// TIA Portal V16 export
// export: Created 2022-11-17T15:49:26.75894Z, ExportSetting WithDefaults, DisplayName Totally Integrated Automation Portal, DisplayVersion V16 Update 6, DisplayName TIA Portal Version Control Interface, DisplayVersion V16 Update 2, DisplayName TIA Portal Openness, DisplayVersion V16 Update 6, DisplayName SINAMICS Startdrive Advanced, DisplayVersion V16 Update 5, DisplayName SINAMICS Startdrive G130, G150, S120, S150, SINAMICS MV, S210, DisplayVersion V16 Update 5, DisplayName SINAMICS Startdrive G110M, G120, G120C, G120D, G120P, G115D, DisplayVersion V16 Update 5, DisplayName STEP 7 Professional, DisplayVersion V16 Update 6, DisplayName STEP 7 Safety, DisplayVersion V16, DisplayName WinCC Advanced, DisplayVersion V16 Update 6
FUNCTION "FC58_TableRotationPos" : Void   // FC58, LAD
{ S7_Optimized_Access := 'FALSE' }
VERSION : 0.1
// stored: AutoNumber false, IsIECCheckEnabled false, SetENOAutomatically false, UDAEnableTagReadback false
   VAR_INPUT
      PHASE : Bool;
   END_VAR
   VAR_TEMP
      TempDInt3 : DInt;
      PulseOffset : DInt;
      AC1 : Real;
      AC2 : Real;
      AC3 : Real;
      DeltaV : Real;
      DeltaVMax : Real;
      VattpiuVmin : Real;
      VmaxpiuVmin : Real;
      AC1_INT : Int;
      PulseReset : Bool;
      TEMPOMAX : Real;
      TEMPO : Real;
      Encoder : Int;
      TempDint : DInt;
      TempInt : Int;
      TempDint2 : DInt;
      TempDInt4 : DInt;
      TempWord : Word;
   END_VAR
   VAR_TEMP   // added for the SCL form of the ladder/FBD networks
      _w1 : Bool;
   END_VAR
BEGIN

REGION Network 1
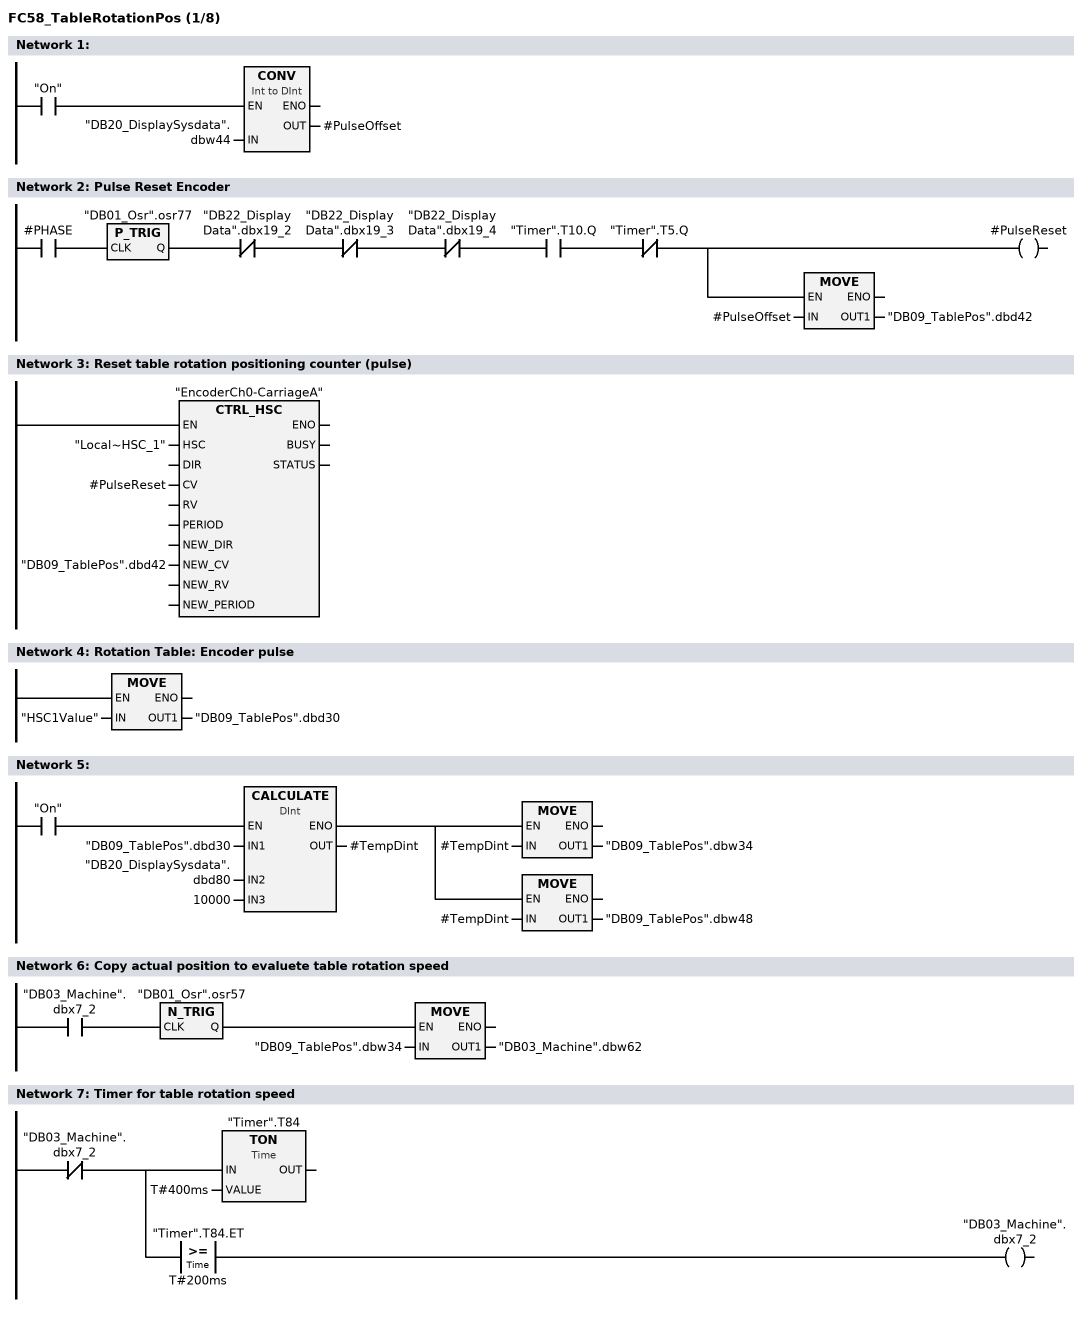
   RUNG wire#powerrail
      Contact( "On" )
      { S7_Templates := "[SrcType := Int, DestType := DInt]"; S7_GenerateENO := "TRUE" } Convert(in := "DB20_DisplaySysdata".dbw44, out => #PulseOffset)
   END_RUNG
   // the same network as SCL:
   IF "On" THEN #PulseOffset := INT_TO_DINT("DB20_DisplaySysdata".dbw44); END_IF;
END_REGION

REGION Network 2: Pulse Reset Encoder
   RUNG wire#powerrail
      Contact( #PHASE )
      P_Trig( "DB01_Osr".osr77 )
      I_Contact( "DB22_DisplayData".dbx19_2 )
      I_Contact( "DB22_DisplayData".dbx19_3 )
      I_Contact( "DB22_DisplayData".dbx19_4 )
      Contact( "Timer".T10.Q )
      I_Contact( "Timer".T5.Q )
      wire#w1
      Coil( #PulseReset )
   END_RUNG
   RUNG wire#w1
      { S7_GenerateENO := "TRUE" } Move(in := #PulseOffset, out1 => "DB09_TablePos".dbd42)
   END_RUNG
   // the same network as SCL:
   #_w1 := #PHASE AND NOT "DB01_Osr".osr77;   // rising edge
   "DB01_Osr".osr77 := #PHASE;
   #PulseReset := #_w1 AND NOT "DB22_DisplayData".dbx19_2 AND NOT "DB22_DisplayData".dbx19_3 AND NOT "DB22_DisplayData".dbx19_4 AND "Timer".T10.Q AND NOT "Timer".T5.Q;
   IF #PulseReset THEN "DB09_TablePos".dbd42 := #PulseOffset; END_IF;
END_REGION

REGION Network 3: Reset table rotation positioning counter (pulse)
   RUNG wire#powerrail
      "EncoderCh0-CarriageA".CTRL_HSC(HSC := "Local~HSC_1", DIR :=, CV := #PulseReset, RV :=, PERIOD :=, NEW_DIR :=, NEW_CV := "DB09_TablePos".dbd42, NEW_RV :=, NEW_PERIOD :=, BUSY =>, STATUS =>)
   END_RUNG
   // the same network as SCL:
   "EncoderCh0-CarriageA"(HSC := "Local~HSC_1", CV := #PulseReset, NEW_CV := "DB09_TablePos".dbd42);   // CTRL_HSC
END_REGION

REGION Network 4: Rotation Table: Encoder pulse
   RUNG wire#powerrail
      { S7_GenerateENO := "TRUE" } Move(in := "HSC1Value", out1 => "DB09_TablePos".dbd30)
   END_RUNG
   // the same network as SCL:
   "DB09_TablePos".dbd30 := "HSC1Value";
END_REGION

REGION Network 5
   RUNG wire#powerrail
      Contact( "On" )
      { S7_Templates := "SrcType := DInt"; S7_GenerateENO := "TRUE"; S7_Expression := "((In1*In2)/In3)" } Calculate(in1 := "DB09_TablePos".dbd30, in2 := "DB20_DisplaySysdata".dbd80, in3 := 10000, out => #TempDint)
      wire#w1
      { S7_GenerateENO := "TRUE" } Move(in := #TempDint, out1 => "DB09_TablePos".dbw34)
   END_RUNG
   RUNG wire#w1
      { S7_GenerateENO := "TRUE" } Move(in := #TempDint, out1 => "DB09_TablePos".dbw48)
   END_RUNG
   // the same network as SCL:
   // ENO of a box is taken as its EN; it also drops when the box reports an error
   IF "On" THEN
       #TempDint := (("DB09_TablePos".dbd30*"DB20_DisplaySysdata".dbd80)/10000);
       "DB09_TablePos".dbw34 := #TempDint;
       "DB09_TablePos".dbw48 := #TempDint;
   END_IF;
END_REGION

REGION Network 6: Copy actual position to evaluete table rotation speed
   RUNG wire#powerrail
      Contact( "DB03_Machine".dbx7_2 )
      N_Trig( "DB01_Osr".osr57 )
      { S7_GenerateENO := "TRUE" } Move(in := "DB09_TablePos".dbw34, out1 => "DB03_Machine".dbw62)
   END_RUNG
   // the same network as SCL:
   #_w1 := NOT "DB03_Machine".dbx7_2 AND "DB01_Osr".osr57;   // falling edge
   "DB01_Osr".osr57 := "DB03_Machine".dbx7_2;
   IF #_w1 THEN "DB03_Machine".dbw62 := "DB09_TablePos".dbw34; END_IF;
END_REGION

REGION Network 7: Timer for table rotation speed
   #_w1 := NOT "DB03_Machine".dbx7_2;
   "Timer".T84.TON(IN := #_w1, PT := T#400ms);   // TON coil
   "DB03_Machine".dbx7_2 := #_w1 AND ("Timer".T84.ET >= T#200ms);
END_REGION

REGION Network 8: Speed calculation (1)
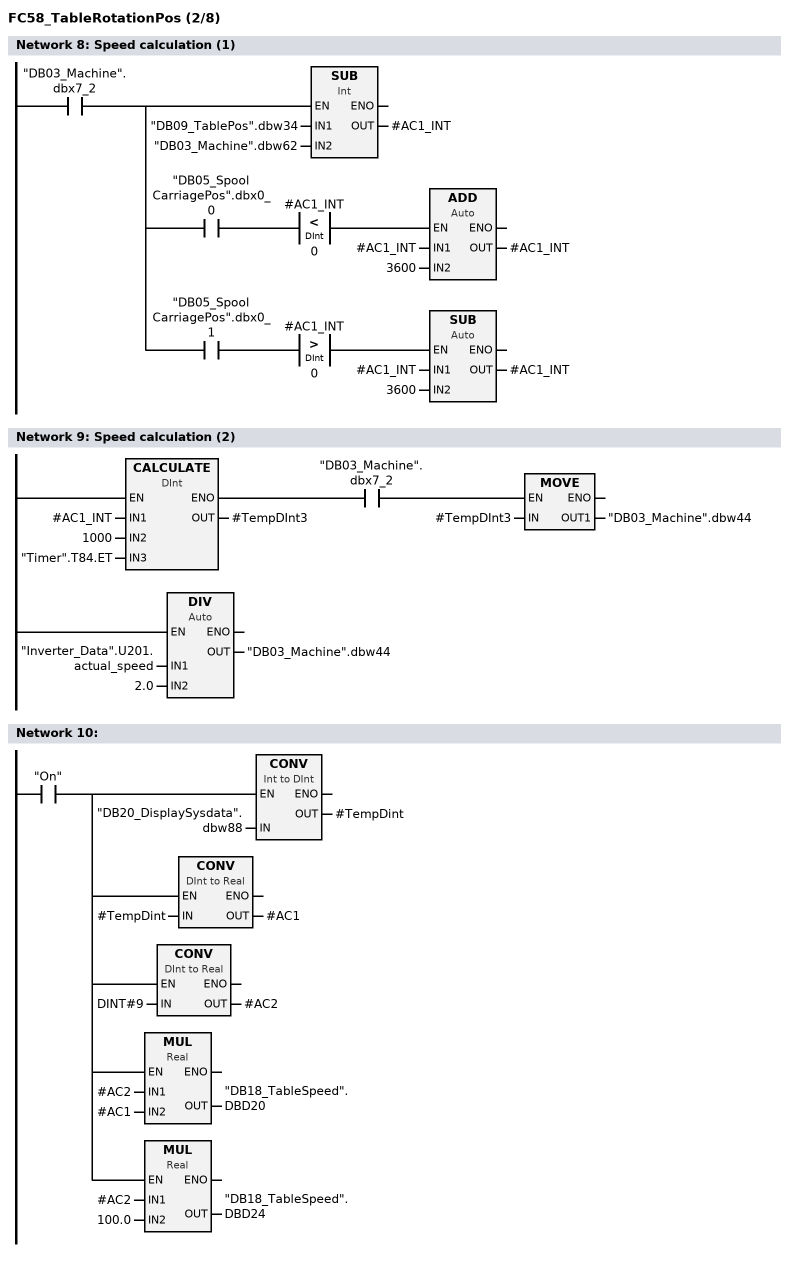
   RUNG wire#powerrail
      Contact( "DB03_Machine".dbx7_2 )
      wire#w1
      { S7_Templates := "SrcType := Int"; S7_GenerateENO := "TRUE" } Sub(in1 := "DB09_TablePos".dbw34, in2 := "DB03_Machine".dbw62, out => #AC1_INT)
   END_RUNG
   RUNG wire#w1
      Contact( "DB05_SpoolCarriagePos".dbx0_0 )
      { S7_Templates := "SrcType := DInt" } LT_Contact(in1 := #AC1_INT, in2 := 0)
      { S7_GenerateENO := "TRUE" } Add(in1 := #AC1_INT, in2 := 3600, out => #AC1_INT)
   END_RUNG
   RUNG wire#w1
      Contact( "DB05_SpoolCarriagePos".dbx0_1 )
      { S7_Templates := "SrcType := DInt" } GT_Contact(in1 := #AC1_INT, in2 := 0)
      { S7_GenerateENO := "TRUE" } Sub(in1 := #AC1_INT, in2 := 3600, out => #AC1_INT)
   END_RUNG
   // the same network as SCL:
   IF "DB03_Machine".dbx7_2 THEN #AC1_INT := "DB09_TablePos".dbw34 - "DB03_Machine".dbw62; END_IF;
   IF "DB03_Machine".dbx7_2 AND "DB05_SpoolCarriagePos".dbx0_0 AND (#AC1_INT < 0) THEN
       #AC1_INT := #AC1_INT + 3600;
   END_IF;
   IF "DB03_Machine".dbx7_2 AND "DB05_SpoolCarriagePos".dbx0_1 AND (#AC1_INT > 0) THEN
       #AC1_INT := #AC1_INT - 3600;
   END_IF;
END_REGION

REGION Network 9: Speed calculation (2)
   RUNG wire#powerrail
      { S7_Templates := "SrcType := DInt"; S7_GenerateENO := "TRUE"; S7_Expression := "((In1*In2)/In3)" } Calculate(in1 := #AC1_INT, in2 := 1000, in3 := "Timer".T84.ET, out => #TempDInt3)
      Contact( "DB03_Machine".dbx7_2 )
      { S7_GenerateENO := "TRUE" } Move(in := #TempDInt3, out1 => "DB03_Machine".dbw44)
   END_RUNG
   RUNG wire#powerrail
      Div(in1 := "Inverter_Data".U201.actual_speed, in2 := 2.0, out => "DB03_Machine".dbw44)
   END_RUNG
   // the same network as SCL:
   // ENO of a box is taken as its EN; it also drops when the box reports an error
   #TempDInt3 := ((#AC1_INT*1000)/"Timer".T84.ET);
   IF "DB03_Machine".dbx7_2 THEN "DB03_Machine".dbw44 := #TempDInt3; END_IF;
   "DB03_Machine".dbw44 := "Inverter_Data".U201.actual_speed / 2.0;
END_REGION

REGION Network 10
   RUNG wire#powerrail
      Contact( "On" )
      wire#w1
      { S7_Templates := "[SrcType := Int, DestType := DInt]"; S7_GenerateENO := "TRUE" } Convert(in := "DB20_DisplaySysdata".dbw88, out => #TempDint)
   END_RUNG
   RUNG wire#w1
      { S7_Templates := "[SrcType := DInt, DestType := Real]"; S7_GenerateENO := "TRUE" } Convert(in := #TempDint, out => #AC1)
   END_RUNG
   RUNG wire#w1
      { S7_Templates := "[SrcType := DInt, DestType := Real]"; S7_GenerateENO := "TRUE" } Convert(in := DINT#9, out => #AC2)
   END_RUNG
   RUNG wire#w1
      { S7_Templates := "SrcType := Real"; S7_GenerateENO := "TRUE" } Mul(in1 := #AC2, in2 := #AC1, out => "DB18_TableSpeed".DBD20)
   END_RUNG
   RUNG wire#w1
      { S7_Templates := "SrcType := Real"; S7_GenerateENO := "TRUE" } Mul(in1 := #AC2, in2 := 100.0, out => "DB18_TableSpeed".DBD24)
   END_RUNG
   // the same network as SCL:
   IF "On" THEN
       #TempDint := INT_TO_DINT("DB20_DisplaySysdata".dbw88);
       #AC1 := DINT_TO_REAL(#TempDint);
       #AC2 := DINT_TO_REAL(DINT#9);
       "DB18_TableSpeed".DBD20 := #AC2 * #AC1;
       "DB18_TableSpeed".DBD24 := #AC2 * 100.0;
   END_IF;
END_REGION

REGION Network 11
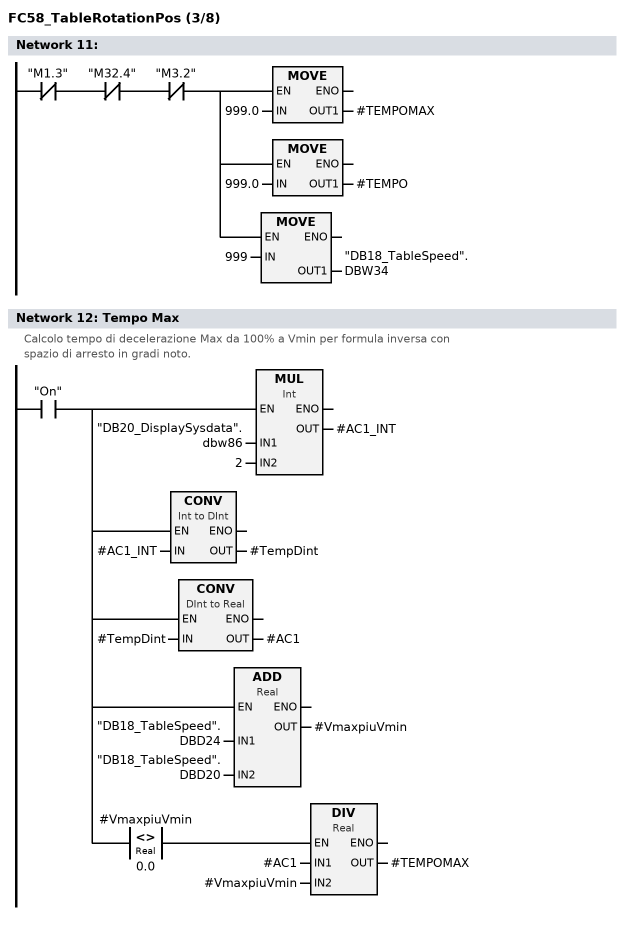
   RUNG wire#powerrail
      I_Contact( "M1.3" )
      I_Contact( "M32.4" )
      I_Contact( "M3.2" )
      wire#w1
      { S7_GenerateENO := "TRUE" } Move(in := 999.0, out1 => #TEMPOMAX)
   END_RUNG
   RUNG wire#w1
      { S7_GenerateENO := "TRUE" } Move(in := 999.0, out1 => #TEMPO)
   END_RUNG
   RUNG wire#w1
      { S7_GenerateENO := "TRUE" } Move(in := 999, out1 => "DB18_TableSpeed".DBW34)
   END_RUNG
   // the same network as SCL:
   IF NOT "M1.3" AND NOT "M32.4" AND NOT "M3.2" THEN
       #TEMPOMAX := 999.0;
       #TEMPO := 999.0;
       "DB18_TableSpeed".DBW34 := 999;
   END_IF;
END_REGION

REGION Network 12: Tempo Max
   // Calcolo tempo di decelerazione Max da 100% a Vmin per formula inversa con 
   // spazio di arresto in gradi noto.
   RUNG wire#powerrail
      Contact( "On" )
      wire#w1
      { S7_Templates := "SrcType := Int"; S7_GenerateENO := "TRUE" } Mul(in1 := "DB20_DisplaySysdata".dbw86, in2 := 2, out => #AC1_INT)
   END_RUNG
   RUNG wire#w1
      { S7_Templates := "[SrcType := Int, DestType := DInt]"; S7_GenerateENO := "TRUE" } Convert(in := #AC1_INT, out => #TempDint)
   END_RUNG
   RUNG wire#w1
      { S7_Templates := "[SrcType := DInt, DestType := Real]"; S7_GenerateENO := "TRUE" } Convert(in := #TempDint, out => #AC1)
   END_RUNG
   RUNG wire#w1
      { S7_Templates := "SrcType := Real"; S7_GenerateENO := "TRUE" } Add(in1 := "DB18_TableSpeed".DBD24, in2 := "DB18_TableSpeed".DBD20, out => #VmaxpiuVmin)
   END_RUNG
   RUNG wire#w1
      { S7_Templates := "SrcType := Real" } NE_Contact(in1 := #VmaxpiuVmin, in2 := 0.0)
      { S7_Templates := "SrcType := Real"; S7_GenerateENO := "TRUE" } Div(in1 := #AC1, in2 := #VmaxpiuVmin, out => #TEMPOMAX)
   END_RUNG
   // the same network as SCL:
   IF "On" THEN
       #AC1_INT := "DB20_DisplaySysdata".dbw86 * 2;
       #TempDint := INT_TO_DINT(#AC1_INT);
       #AC1 := DINT_TO_REAL(#TempDint);
       #VmaxpiuVmin := "DB18_TableSpeed".DBD24 + "DB18_TableSpeed".DBD20;
   END_IF;
   IF "On" AND (#VmaxpiuVmin <> 0.0) THEN #TEMPOMAX := #AC1 / #VmaxpiuVmin; END_IF;
END_REGION

REGION Network 13: Calcolo tempo di decelerazione da Vatt a Vmin per calcolo spazio di arresto
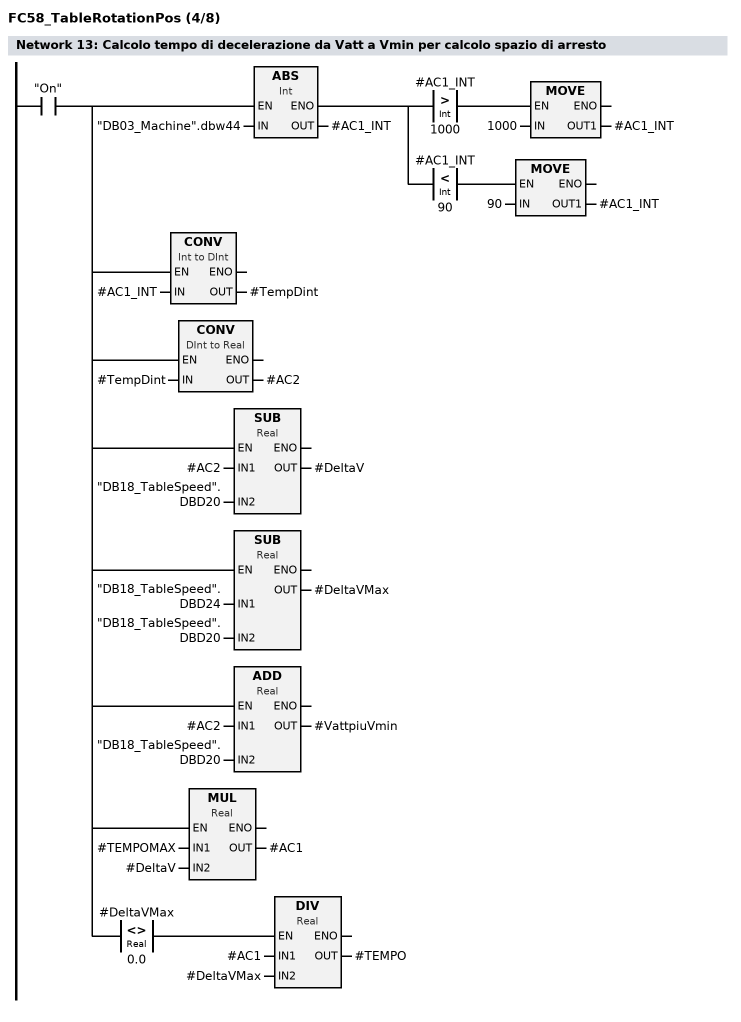
   RUNG wire#powerrail
      Contact( "On" )
      wire#w1
      { S7_Templates := "SrcType := Int" } Abs(in := "DB03_Machine".dbw44, out => #AC1_INT)
      wire#w2
      { S7_Templates := "SrcType := Int" } GT_Contact(in1 := #AC1_INT, in2 := 1000)
      Move(in := 1000, out1 => #AC1_INT)
   END_RUNG
   RUNG wire#w2
      { S7_Templates := "SrcType := Int" } LT_Contact(in1 := #AC1_INT, in2 := 90)
      Move(in := 90, out1 => #AC1_INT)
   END_RUNG
   RUNG wire#w1
      { S7_Templates := "[SrcType := Int, DestType := DInt]"; S7_GenerateENO := "TRUE" } Convert(in := #AC1_INT, out => #TempDint)
   END_RUNG
   RUNG wire#w1
      { S7_Templates := "[SrcType := DInt, DestType := Real]"; S7_GenerateENO := "TRUE" } Convert(in := #TempDint, out => #AC2)
   END_RUNG
   RUNG wire#w1
      { S7_Templates := "SrcType := Real"; S7_GenerateENO := "TRUE" } Sub(in1 := #AC2, in2 := "DB18_TableSpeed".DBD20, out => #DeltaV)
   END_RUNG
   RUNG wire#w1
      { S7_Templates := "SrcType := Real"; S7_GenerateENO := "TRUE" } Sub(in1 := "DB18_TableSpeed".DBD24, in2 := "DB18_TableSpeed".DBD20, out => #DeltaVMax)
   END_RUNG
   RUNG wire#w1
      { S7_Templates := "SrcType := Real"; S7_GenerateENO := "TRUE" } Add(in1 := #AC2, in2 := "DB18_TableSpeed".DBD20, out => #VattpiuVmin)
   END_RUNG
   RUNG wire#w1
      { S7_Templates := "SrcType := Real"; S7_GenerateENO := "TRUE" } Mul(in1 := #TEMPOMAX, in2 := #DeltaV, out => #AC1)
   END_RUNG
   RUNG wire#w1
      { S7_Templates := "SrcType := Real" } NE_Contact(in1 := #DeltaVMax, in2 := 0.0)
      { S7_Templates := "SrcType := Real"; S7_GenerateENO := "TRUE" } Div(in1 := #AC1, in2 := #DeltaVMax, out => #TEMPO)
   END_RUNG
   // the same network as SCL:
   IF "On" THEN #AC1_INT := ABS("DB03_Machine".dbw44); END_IF;
   IF "On" AND (#AC1_INT > 1000) THEN #AC1_INT := 1000; END_IF;
   IF "On" AND (#AC1_INT < 90) THEN #AC1_INT := 90; END_IF;
   IF "On" THEN
       #TempDint := INT_TO_DINT(#AC1_INT);
       #AC2 := DINT_TO_REAL(#TempDint);
       #DeltaV := #AC2 - "DB18_TableSpeed".DBD20;
       #DeltaVMax := "DB18_TableSpeed".DBD24 - "DB18_TableSpeed".DBD20;
       #VattpiuVmin := #AC2 + "DB18_TableSpeed".DBD20;
       #AC1 := #TEMPOMAX * #DeltaV;
   END_IF;
   IF "On" AND (#DeltaVMax <> 0.0) THEN #TEMPO := #AC1 / #DeltaVMax; END_IF;
END_REGION

REGION Network 14: Decelerazione
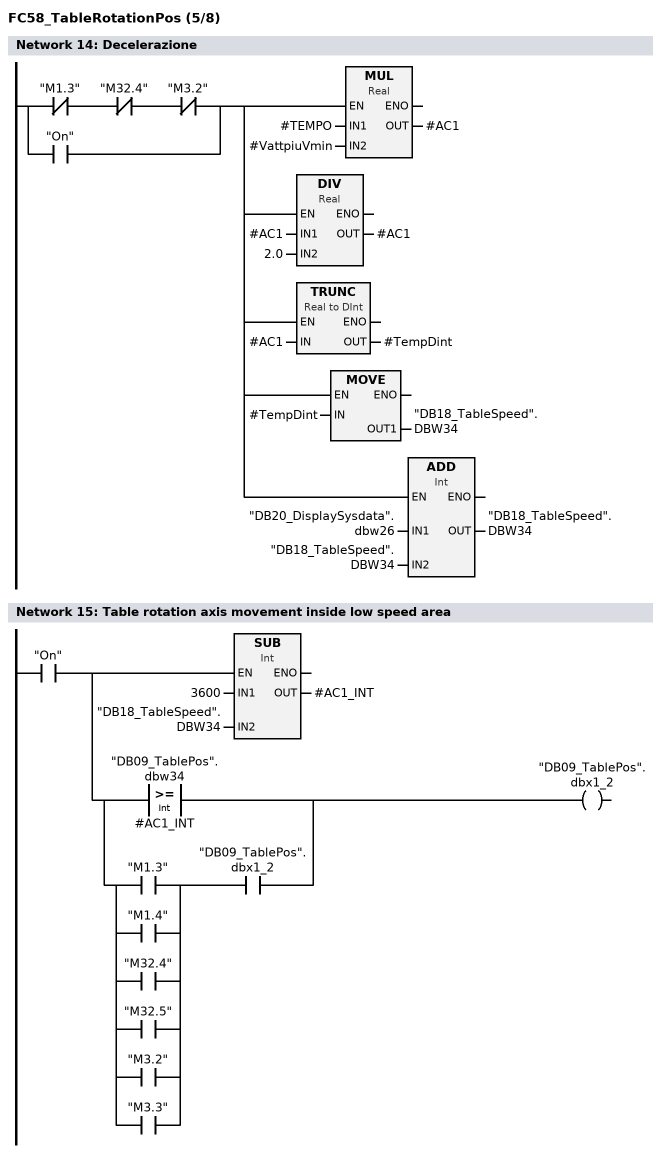
   RUNG wire#powerrail
      I_Contact( "M1.3" )
      I_Contact( "M32.4" )
      I_Contact( "M3.2" )
      wire#w1
      { S7_Templates := "SrcType := Real"; S7_GenerateENO := "TRUE" } Mul(in1 := #TEMPO, in2 := #VattpiuVmin, out => #AC1)
   END_RUNG
   RUNG wire#powerrail
      Contact( "On" )
   END_RUNG wire#w1
   RUNG wire#w1
      { S7_Templates := "SrcType := Real"; S7_GenerateENO := "TRUE" } Div(in1 := #AC1, in2 := 2.0, out => #AC1)
   END_RUNG
   RUNG wire#w1
      { S7_Templates := "[SrcType := Real, DestType := DInt]"; S7_GenerateENO := "TRUE" } Trunc(in := #AC1, out => #TempDint)
   END_RUNG
   RUNG wire#w1
      { S7_GenerateENO := "TRUE" } Move(in := #TempDint, out1 => "DB18_TableSpeed".DBW34)
   END_RUNG
   RUNG wire#w1
      { S7_Templates := "SrcType := Int"; S7_GenerateENO := "TRUE" } Add(in1 := "DB20_DisplaySysdata".dbw26, in2 := "DB18_TableSpeed".DBW34, out => "DB18_TableSpeed".DBW34)
   END_RUNG
   // the same network as SCL:
   IF (NOT "M1.3" AND NOT "M32.4" AND NOT "M3.2") OR "On" THEN
       #AC1 := #TEMPO * #VattpiuVmin;
       #AC1 := #AC1 / 2.0;
       #TempDint := TRUNC(#AC1);
       "DB18_TableSpeed".DBW34 := #TempDint;
       "DB18_TableSpeed".DBW34 := "DB20_DisplaySysdata".dbw26 + "DB18_TableSpeed".DBW34;
   END_IF;
END_REGION

REGION Network 15: Table rotation axis movement inside low speed area
   RUNG wire#powerrail
      Contact( "On" )
      wire#w1
      { S7_Templates := "SrcType := Int"; S7_GenerateENO := "TRUE" } Sub(in1 := 3600, in2 := "DB18_TableSpeed".DBW34, out => #AC1_INT)
   END_RUNG
   RUNG wire#w1
      { S7_Templates := "SrcType := Int" } GE_Contact(in1 := "DB09_TablePos".dbw34, in2 := #AC1_INT)
      wire#w2
      Coil( "DB09_TablePos".dbx1_2 )
   END_RUNG
   RUNG wire#w1
      Contact( "M1.3" )
      wire#w3
      Contact( "DB09_TablePos".dbx1_2 )
   END_RUNG wire#w2
   RUNG wire#w1
      Contact( "M1.4" )
   END_RUNG wire#w3
   RUNG wire#w1
      Contact( "M32.4" )
   END_RUNG wire#w3
   RUNG wire#w1
      Contact( "M32.5" )
   END_RUNG wire#w3
   RUNG wire#w1
      Contact( "M3.2" )
   END_RUNG wire#w3
   RUNG wire#w1
      Contact( "M3.3" )
   END_RUNG wire#w3
   // the same network as SCL:
   IF "On" THEN #AC1_INT := 3600 - "DB18_TableSpeed".DBW34; END_IF;
   "DB09_TablePos".dbx1_2 := "On" AND (("DB09_TablePos".dbw34 >= #AC1_INT) OR (("M1.3" OR "M1.4" OR "M32.4" OR "M32.5" OR "M3.2" OR "M3.3") AND "DB09_TablePos".dbx1_2));
END_REGION

REGION Network 16: Table rotation position loading/Unloading
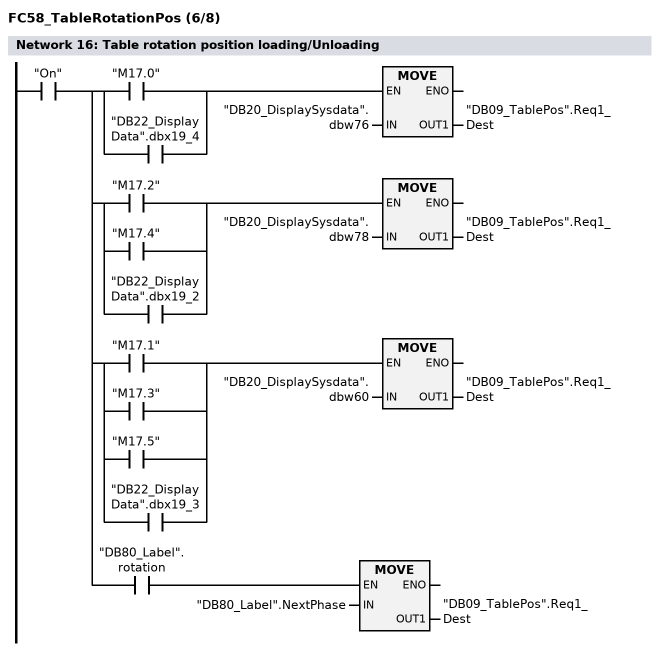
   RUNG wire#powerrail
      Contact( "On" )
      wire#w1
      Contact( "M17.0" )
      wire#w2
      { S7_GenerateENO := "TRUE" } Move(in := "DB20_DisplaySysdata".dbw76, out1 => "DB09_TablePos".Req1_Dest)
   END_RUNG
   RUNG wire#w1
      Contact( "DB22_DisplayData".dbx19_4 )
   END_RUNG wire#w2
   RUNG wire#w1
      Contact( "M17.2" )
      wire#w3
      { S7_GenerateENO := "TRUE" } Move(in := "DB20_DisplaySysdata".dbw78, out1 => "DB09_TablePos".Req1_Dest)
   END_RUNG
   RUNG wire#w1
      Contact( "M17.4" )
   END_RUNG wire#w3
   RUNG wire#w1
      Contact( "DB22_DisplayData".dbx19_2 )
   END_RUNG wire#w3
   RUNG wire#w1
      Contact( "M17.1" )
      wire#w4
      { S7_GenerateENO := "TRUE" } Move(in := "DB20_DisplaySysdata".dbw60, out1 => "DB09_TablePos".Req1_Dest)
   END_RUNG
   RUNG wire#w1
      Contact( "M17.3" )
   END_RUNG wire#w4
   RUNG wire#w1
      Contact( "M17.5" )
   END_RUNG wire#w4
   RUNG wire#w1
      Contact( "DB22_DisplayData".dbx19_3 )
   END_RUNG wire#w4
   RUNG wire#w1
      Contact( "DB80_Label".rotation )
      { S7_GenerateENO := "TRUE" } Move(in := "DB80_Label".NextPhase, out1 => "DB09_TablePos".Req1_Dest)
   END_RUNG
   // the same network as SCL:
   IF "On" AND ("M17.0" OR "DB22_DisplayData".dbx19_4) THEN
       "DB09_TablePos".Req1_Dest := "DB20_DisplaySysdata".dbw76;
   END_IF;
   IF "On" AND ("M17.2" OR "M17.4" OR "DB22_DisplayData".dbx19_2) THEN
       "DB09_TablePos".Req1_Dest := "DB20_DisplaySysdata".dbw78;
   END_IF;
   IF "On" AND ("M17.1" OR "M17.3" OR "M17.5" OR "DB22_DisplayData".dbx19_3) THEN
       "DB09_TablePos".Req1_Dest := "DB20_DisplaySysdata".dbw60;
   END_IF;
   IF "On" AND "DB80_Label".rotation THEN "DB09_TablePos".Req1_Dest := "DB80_Label".NextPhase; END_IF;
END_REGION

REGION Network 17
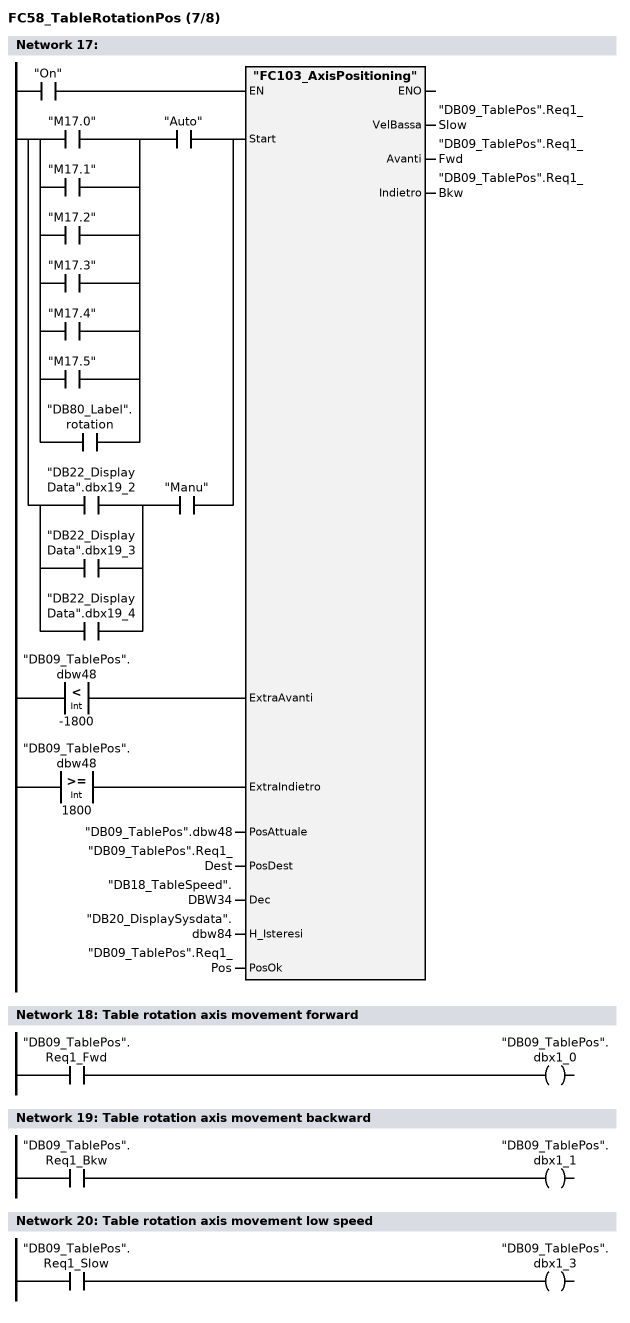
   RUNG wire#powerrail
      Contact( "On" )
      "FC103_AxisPositioning"(Start := wire#w3, ExtraAvanti := wire#w4, ExtraIndietro := wire#w5, PosAttuale := "DB09_TablePos".dbw48, PosDest := "DB09_TablePos".Req1_Dest, Dec := "DB18_TableSpeed".DBW34, H_Isteresi := "DB20_DisplaySysdata".dbw84, PosOk := "DB09_TablePos".Req1_Pos, VelBassa => "DB09_TablePos".Req1_Slow, Avanti => "DB09_TablePos".Req1_Fwd, Indietro => "DB09_TablePos".Req1_Bkw)
   END_RUNG
   RUNG wire#powerrail
      Contact( "M17.0" )
      wire#w1
      Contact( "Auto" )
   END_RUNG wire#w3
   RUNG wire#powerrail
      Contact( "M17.1" )
   END_RUNG wire#w1
   RUNG wire#powerrail
      Contact( "M17.2" )
   END_RUNG wire#w1
   RUNG wire#powerrail
      Contact( "M17.3" )
   END_RUNG wire#w1
   RUNG wire#powerrail
      Contact( "M17.4" )
   END_RUNG wire#w1
   RUNG wire#powerrail
      Contact( "M17.5" )
   END_RUNG wire#w1
   RUNG wire#powerrail
      Contact( "DB80_Label".rotation )
   END_RUNG wire#w1
   RUNG wire#powerrail
      Contact( "DB22_DisplayData".dbx19_2 )
      wire#w2
      Contact( "Manu" )
   END_RUNG wire#w3
   RUNG wire#powerrail
      Contact( "DB22_DisplayData".dbx19_3 )
   END_RUNG wire#w2
   RUNG wire#powerrail
      Contact( "DB22_DisplayData".dbx19_4 )
   END_RUNG wire#w2
   RUNG wire#powerrail
      { S7_Templates := "SrcType := Int" } LT_Contact(in1 := "DB09_TablePos".dbw48, in2 := -1800)
   END_RUNG wire#w4
   RUNG wire#powerrail
      { S7_Templates := "SrcType := Int" } GE_Contact(in1 := "DB09_TablePos".dbw48, in2 := 1800)
   END_RUNG wire#w5
   // the same network as SCL:
   IF "On" THEN
       "FC103_AxisPositioning"(Start := (("M17.0" OR "M17.1" OR "M17.2" OR "M17.3" OR "M17.4" OR "M17.5" OR "DB80_Label".rotation) AND "Auto") OR (("DB22_DisplayData".dbx19_2 OR "DB22_DisplayData".dbx19_3 OR "DB22_DisplayData".dbx19_4) AND "Manu"),
                               ExtraAvanti := "DB09_TablePos".dbw48 < (-1800),
                               ExtraIndietro := "DB09_TablePos".dbw48 >= 1800,
                               PosAttuale := "DB09_TablePos".dbw48,
                               PosDest := "DB09_TablePos".Req1_Dest,
                               Dec := "DB18_TableSpeed".DBW34,
                               H_Isteresi := "DB20_DisplaySysdata".dbw84,
                               PosOk := "DB09_TablePos".Req1_Pos,
                               VelBassa => "DB09_TablePos".Req1_Slow,
                               Avanti => "DB09_TablePos".Req1_Fwd,
                               Indietro => "DB09_TablePos".Req1_Bkw);
   END_IF;
END_REGION

REGION Network 18: Table rotation axis movement forward
   RUNG wire#powerrail
      Contact( "DB09_TablePos".Req1_Fwd )
      Coil( "DB09_TablePos".dbx1_0 )
   END_RUNG
   // the same network as SCL:
   "DB09_TablePos".dbx1_0 := "DB09_TablePos".Req1_Fwd;
END_REGION

REGION Network 19: Table rotation axis movement backward
   RUNG wire#powerrail
      Contact( "DB09_TablePos".Req1_Bkw )
      Coil( "DB09_TablePos".dbx1_1 )
   END_RUNG
   // the same network as SCL:
   "DB09_TablePos".dbx1_1 := "DB09_TablePos".Req1_Bkw;
END_REGION

REGION Network 20: Table rotation axis movement low speed
   RUNG wire#powerrail
      Contact( "DB09_TablePos".Req1_Slow )
      Coil( "DB09_TablePos".dbx1_3 )
   END_RUNG
   // the same network as SCL:
   "DB09_TablePos".dbx1_3 := "DB09_TablePos".Req1_Slow;
END_REGION

REGION Network 21: TABLE ENCODER CHECK
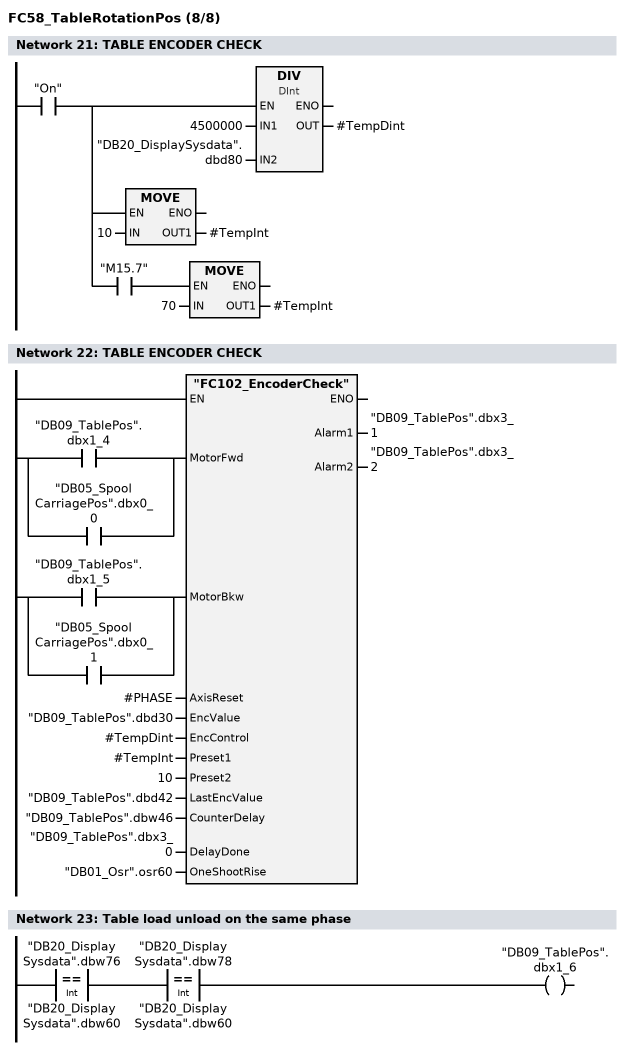
   RUNG wire#powerrail
      Contact( "On" )
      wire#w1
      { S7_Templates := "SrcType := DInt"; S7_GenerateENO := "TRUE" } Div(in1 := 4500000, in2 := "DB20_DisplaySysdata".dbd80, out => #TempDint)
   END_RUNG
   RUNG wire#w1
      { S7_GenerateENO := "TRUE" } Move(in := 10, out1 => #TempInt)
   END_RUNG
   RUNG wire#w1
      Contact( "M15.7" )
      { S7_GenerateENO := "TRUE" } Move(in := 70, out1 => #TempInt)
   END_RUNG
   // the same network as SCL:
   IF "On" THEN
       #TempDint := 4500000 / "DB20_DisplaySysdata".dbd80;
       #TempInt := 10;
   END_IF;
   IF "On" AND "M15.7" THEN #TempInt := 70; END_IF;
END_REGION

REGION Network 22: TABLE ENCODER CHECK
   RUNG wire#powerrail
      "FC102_EncoderCheck"(MotorFwd := wire#w1, MotorBkw := wire#w2, AxisReset := #PHASE, EncValue := "DB09_TablePos".dbd30, EncControl := #TempDint, Preset1 := #TempInt, Preset2 := 10, LastEncValue := "DB09_TablePos".dbd42, CounterDelay := "DB09_TablePos".dbw46, DelayDone := "DB09_TablePos".dbx3_0, OneShootRise := "DB01_Osr".osr60, Alarm1 => "DB09_TablePos".dbx3_1, Alarm2 => "DB09_TablePos".dbx3_2)
   END_RUNG
   RUNG wire#powerrail
      Contact( "DB09_TablePos".dbx1_4 )
   END_RUNG wire#w1
   RUNG wire#powerrail
      Contact( "DB05_SpoolCarriagePos".dbx0_0 )
   END_RUNG wire#w1
   RUNG wire#powerrail
      Contact( "DB09_TablePos".dbx1_5 )
   END_RUNG wire#w2
   RUNG wire#powerrail
      Contact( "DB05_SpoolCarriagePos".dbx0_1 )
   END_RUNG wire#w2
   // the same network as SCL:
   "FC102_EncoderCheck"(MotorFwd := "DB09_TablePos".dbx1_4 OR "DB05_SpoolCarriagePos".dbx0_0,
                        MotorBkw := "DB09_TablePos".dbx1_5 OR "DB05_SpoolCarriagePos".dbx0_1,
                        AxisReset := #PHASE,
                        EncValue := "DB09_TablePos".dbd30,
                        EncControl := #TempDint,
                        Preset1 := #TempInt,
                        Preset2 := 10,
                        LastEncValue := "DB09_TablePos".dbd42,
                        CounterDelay := "DB09_TablePos".dbw46,
                        DelayDone := "DB09_TablePos".dbx3_0,
                        OneShootRise := "DB01_Osr".osr60,
                        Alarm1 => "DB09_TablePos".dbx3_1,
                        Alarm2 => "DB09_TablePos".dbx3_2);
END_REGION

REGION Network 23: Table load unload on the same phase
   RUNG wire#powerrail
      { S7_Templates := "SrcType := Int" } EQ_Contact(in1 := "DB20_DisplaySysdata".dbw76, in2 := "DB20_DisplaySysdata".dbw60)
      { S7_Templates := "SrcType := Int" } EQ_Contact(in1 := "DB20_DisplaySysdata".dbw78, in2 := "DB20_DisplaySysdata".dbw60)
      Coil( "DB09_TablePos".dbx1_6 )
   END_RUNG
   // the same network as SCL:
   "DB09_TablePos".dbx1_6 := ("DB20_DisplaySysdata".dbw76 = "DB20_DisplaySysdata".dbw60) AND ("DB20_DisplaySysdata".dbw78 = "DB20_DisplaySysdata".dbw60);
END_REGION
END_FUNCTION
